// TIA Portal V16 export
// export: Created 2026-03-31T12:43:25.3847963Z, ExportSetting WithDefaults, DisplayName Totally Integrated Automation Portal, DisplayVersion V16, DisplayName TIA Portal Version Control Interface, DisplayVersion V16, DisplayName TIA Portal Openness, DisplayVersion V16, DisplayName STEP 7 Professional, DisplayVersion V16, DisplayName STEP 7 Safety, DisplayVersion V16, DisplayName WinCC Advanced, DisplayVersion V16
VAR_GLOBAL   // PLC tag table "Tag table_2"
   Pol_sklad_sens AT %IW40 : Int;
   Pol_sens AT %IW42 : Int;
END_VAR
